// TIA Portal V19 export
TYPE "dtPumpStaging"
   STRUCT
      cmdSmall : Bool := false;
      cmdBig : Bool := false;
      cmdMed : Bool := false;
      tDelay : Time := T#20s;   // 1=P44_05, 2=P44_06
      stageUpThr : Real := 95.0;
      stageDnThr : Real := 45.0;
      activeBig : Int := 0;
   END_STRUCT;
END_TYPE
